// TIA Portal V16 export
// export: Created 2023-10-30T22:43:54.1459984Z, ExportSetting WithDefaults, DisplayName Totally Integrated Automation Portal, DisplayVersion V16, DisplayName TIA Portal Version Control Interface, DisplayVersion V16, DisplayName TIA Portal Openness, DisplayVersion V16, DisplayName SINAMICS Startdrive Advanced, DisplayVersion V16, DisplayName SINAMICS Startdrive G130, G150, S120, S150, SINAMICS MV, S210, DisplayVersion V16, DisplayName SINAMICS Startdrive G110M, G120, G120C, G120D, G120P, DisplayVersion V16, DisplayName STEP 7 Professional, DisplayVersion V16, DisplayName STEP 7 Safety, DisplayVersion V16, DisplayName WinCC Professional, DisplayVersion V16
DATA_BLOCK "MODULO_SECADOR_DB_1"   // DB2
// stored: AutoNumber true, DBAccessibleFromOPCUA true, InstanceOfName MODULO_SECADOR, InstanceOfType FB
"MODULO_SECADOR"
   // VAR_INPUT
   //    Encendido : Bool;
   //    Temperatura : Int;
   //    Humedad : Int;
   //    TempMin : Real;
   //    CtoHR : Real;
   //    PasoCtrlHR : Time;
   // END_VAR
   // VAR_OUTPUT
   //    Actuadores : Bool;
   // END_VAR
   // VAR
   //    Estado : Int;
   //    Timer_FSMHR : Struct
   //       IN : Bool;
   //       PT : Time;
   //       Q : Bool;
   //       ET : Time;
   //    END_STRUCT;
   //    H1 : Real;
   //    H2 : Real;
   //    DH1 : Real;
   //    DH2 : Real;
   //    CRECIMIENTO : Real;
   // END_VAR
BEGIN
END_DATA_BLOCK
